FUNCTION_BLOCK QUERY_GEN (* XML Query Template Generator *)
  (* Standard: 61499 ITA; Function: QUERY Functional Test *)
  (* Version 0.1, 2001-11-27, JHC, Rockwell Automation, Added DSTI, DSTO *)
  (* Version 0.0, 2001-11-24, JHC, Rockwell Automation *)
  (* Compiler header: package fb.rt.ita; *)
  (* Compiler Java IBM VisualAge 3.0 *)
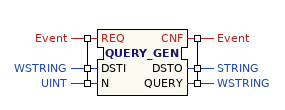
  EVENT_INPUT
    REQ WITH DSTI, N; (* Query Generation Request *)
  END_EVENT
  EVENT_OUTPUT
    CNF WITH DSTO, QUERY; (* Query Generated *)
  END_EVENT
  VAR_INPUT
    DSTI : WSTRING; (* Destination *)
    N : UINT; (* 0=FB,1=Connection *)
  END_VAR
  VAR_OUTPUT
    DSTO : STRING; (* DSTI converted to STRING *)
    QUERY : WSTRING; (* Query Template *)
  END_VAR
END_FUNCTION_BLOCK
